// TIA Portal V17 export
// export: Created 2021-12-03T08:12:47.8881036Z, ExportSetting WithDefaults, DisplayName Totally Integrated Automation Portal, DisplayVersion V17, DisplayName TIA Portal Openness, DisplayVersion V17, DisplayName TIA Portal Version Control Interface, DisplayVersion V17, DisplayName STEP 7 Professional, DisplayVersion V17, DisplayName STEP 7 Safety, DisplayVersion V17, DisplayName WinCC Advanced, DisplayVersion V17
ORGANIZATION_BLOCK "Cyclic_interrupt_100ms"   // OB33, FBD, CyclicInterrupt
TITLE = "Cyclic Interrupt"
VERSION : 0.1
// stored: IsIECCheckEnabled false
   VAR_TEMP
      OB33_EV_CLASS : Byte;   // Bits 0-3 = 1 (Coming event), Bits 4-7 = 1 (Event class 1)
      OB33_STRT_INF : Byte;   // 16#34 (OB 33 has started)
      OB33_PRIORITY : Byte;   // Priority of OB Execution
      OB33_OB_NUMBR : Byte;   // 33 (Organization block 33, OB33)
      OB33_RESERVED_1 : Byte;   // Reserved for system
      OB33_RESERVED_2 : Byte;   // Reserved for system
      OB33_PHS_OFFSET : Int;   // Phase offset (integer, milliseconds)
      OB33_RESERVED_3 : Int;   // Reserved for system
      OB33_EXC_FREQ : Int;   // Frequency of execution (msec)
      OB33_DATE_TIME : Date_And_Time;   // Date and time OB33 started
   END_VAR
BEGIN

REGION Network 2: Always True
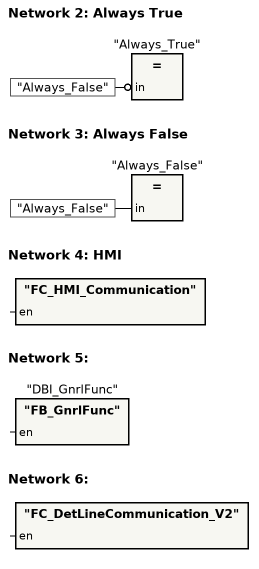
   "Always_True" := NOT "Always_False";
END_REGION

REGION Network 3: Always False
   "Always_False" := "Always_False";
END_REGION

REGION Network 4: HMI
   "FC_HMI_Communication"();
END_REGION

REGION Network 5
   "DBI_GnrlFunc"();   // "FB_GnrlFunc"
END_REGION

REGION Network 6
   "FC_DetLineCommunication_V2"();
END_REGION
END_ORGANIZATION_BLOCK
